PROGRAM P_Warning
VAR
	btRun : BOOL := FALSE;
END_VAR

IF NOT btRun THEN
	ADSLOGSTR(msgCtrlMask := ADSLOG_MSGTYPE_ERROR OR ADSLOG_MSGTYPE_LOG,
			  msgFmtStr := 'hi Thinh',
			  strArg := '');
	btRun := TRUE;
END_IF

END_PROGRAM

(* stored: Version 1.1.0.1, ProductVersion 3.1.4024.12
   POU P_Warning: Id {2d7240f4-6edf-4f06-9bf8-1e28e942cdfe}, SpecialFunc None *)
